FUNCTION_BLOCK New (* _ *)
  (* Version 2015-09-26 *)
END_FUNCTION_BLOCK
(* other elements stored in the file *)
(* SNS LeftPageBorder=-300.0 RightPageBorder=300.0 *)
(* place Diameter=30.0 Name=p1 Num=1 LocNum=1 Mark=1 Clock=0 Capacity=1 Comment=_ *)
(* CommentBox Width=20 Height=20 *)
(* place Diameter=30.0 Name=p2 Num=2 LocNum=2 Mark=0 Clock=0 Capacity=1 Comment=_ *)
(* CommentBox Width=20 Height=20 *)
(* trans Width=30 Height=20 Num=1 LocNum=1 Name=t1 Type=OR TransInscription=_ SwitchMode=s Comment=_ *)
(* CommentBox Width=20 Height=20 *)
(* trans Width=30 Height=20 Num=2 LocNum=2 Name=t2 Type=OR TransInscription=_ SwitchMode=s Comment=_ *)
(* CommentBox Width=20 Height=20 *)
(* trans Width=30 Height=20 Num=3 LocNum=3 Name=t3 Type=OR TransInscription=_ SwitchMode=s Comment=_ *)
(* CommentBox Width=20 Height=20 *)
(* arc StartPoint=t1 EndPoint=p2 ArcWeight=1 Comment=_ *)
(* arc StartPoint=t2 EndPoint=p2 ArcWeight=1 Comment=_ *)
(* arc StartPoint=t3 EndPoint=p2 ArcWeight=1 Comment=_ *)
(* arc StartPoint=p1 EndPoint=t3 ArcWeight=2 Comment=_ *)
(* arc StartPoint=p1 EndPoint=t2 ArcWeight=1 Comment=_ *)
(* arc StartPoint=p1 EndPoint=t1 ArcWeight=2 Comment=_ *)
